PROGRAM PRG_CryoStat
VAR
    fbCRYO_Motor_X : FB_MotionStage;
    fbCRYO_Motor_Y : FB_MotionStage;
    fbCRYO_Motor_Z : FB_MotionStage;
    fbCRYO_Motor_rY : FB_MotionStage;
END_VAR

Main.M22.bHardwareEnable := TRUE;
fbCRYO_Motor_X(stMotionStage:=Main.M22);

Main.M23.bHardwareEnable := TRUE;
fbCRYO_Motor_Y(stMotionStage:=Main.M23);

Main.M24.bHardwareEnable := TRUE;
fbCRYO_Motor_Z(stMotionStage:=Main.M24);

Main.M25.bHardwareEnable := TRUE;
fbCRYO_Motor_rY(stMotionStage:=Main.M25);
Main.M25.bLimitBackwardEnable:=TRUE;
Main.M25.bLimitForwardEnable:=TRUE;

END_PROGRAM

(* stored: Version 1.1.0.1, ProductVersion 3.1.4022.18
   POU PRG_CryoStat: Id {a0ba5752-81fc-458b-b1f7-c5c7a813c6a6}, SpecialFunc None *)
